# EPICS substitutions: gigeApp/Db/tst_gige1.substitutions
#
# gige substitutions file
#

# Generate iocAdmin autosave request
##file autosave_iocAdmin.template
##{
##    {
##        IOC     =   $(IOC)
##    }
##}

# Generate one set per camera
file tst_gige1.template
{
    {   CAM     =   13PS1  }
}
